ABB RobotStudio station: IRB1600_20220617-165440.rsstn

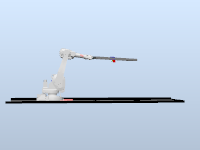
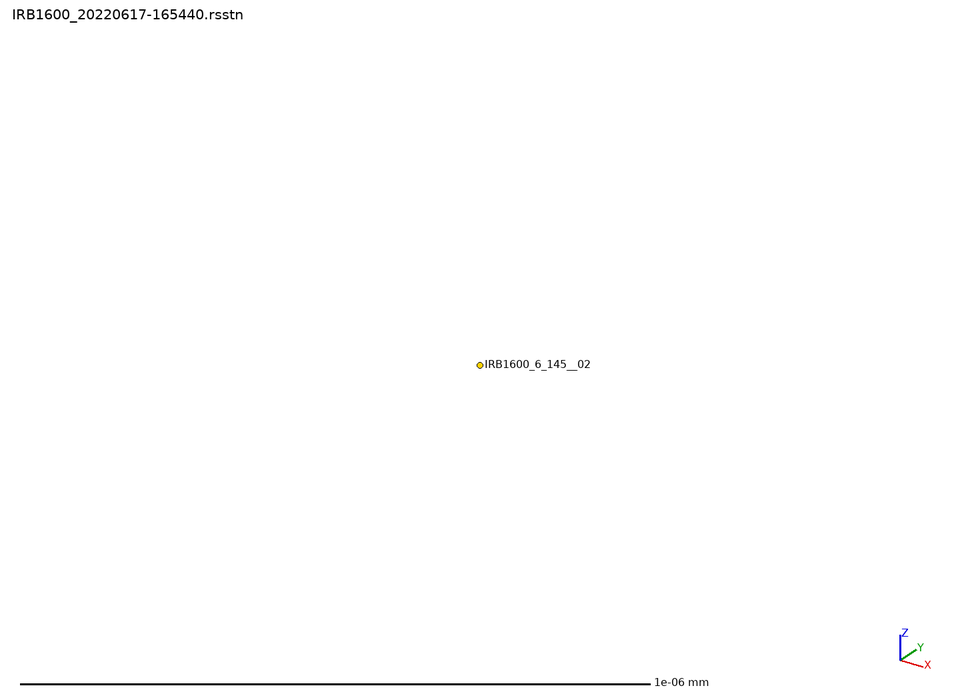
[picture v1: parts stored in the station drawn from their meshes, with robot base, taught points and paths (robot models come from the ABB library and are not in the file)]
Station Solution1 (saved by RobotStudio 22.1.9826.0)
Controller IRB1600_6_145
  mechanical unit ROB_1: IRB1600_6_145__02, 6 joints, base frame (0, 0, 0) mm
Layout (positions relative to the parent item):
  - IRB1600_6_145__02 [mechanism, from Robots\IRB1600_6_145_G_02.rslib] at (0, 0, 0) mm; joint values [0.0015, 0.282, -0.1091, -0.1819, -0.1284, 0.242] (rad or m)
  - flange_connector [part, from Tools\IsoPlate_small_Binzel.rslib] at (1000.78, 2.96, 1052.55) mm, rotated rx 126.74 ry 85.53 rz 128.07 deg
  - plane [part] at (1509.57, 17.68, 1033.56) mm, rotated rx 176.41 ry -2.67 rz -178.59 deg, size 1000 x 1000 x 50 mm
  - Frame_1 [frame]
  - Frame_2 [frame] at (-23.65, -1.83, 250.36) mm
Attachment: flange_connector is attached to IRB1600_6_145__02 / Link6
Attachment: plane is attached to flange_connector
Targets, tools, work objects and paths stored in the station, written as RAPID:
! task T_ROB1
MODULE Module1
  LOCAL PERS wobjdata egm_wobj:=[FALSE,TRUE,"",[[0,0,0],[1,0,0,0]],[[0,0,0],[1,0,0,0]]];
  PROC main()
    ConfJ \On;
  ENDPROC
  PROC EGM_CARTESIAN_MOVE()
    WaitTime 2;
  ENDPROC
  PROC RAPID_MOVE()
  ENDPROC
ENDMODULE

! task T_ROB1
MODULE CalibData
  TASK PERS tooldata Tooldata_4:=[TRUE,[[0,0,0],[1,0,0,0]],[1,[0,0,1],[1,0,0,0],0,0,0]];
  TASK PERS tooldata Tooldata_5:=[TRUE,[[0,0,0],[1,0,0,0]],[1,[0,0,1],[1,0,0,0],0,0,0]];
  TASK PERS tooldata Tooldata_6:=[TRUE,[[0,0,0],[1,0,0,0]],[1,[0,0,1],[1,0,0,0],0,0,0]];
  TASK PERS tooldata Tooldata_7:=[TRUE,[[-23.772999698,2.161000196,740.120999999],[0.707106781,0,-0.707106781,0]],[1,[0,0,1],[1,0,0,0],0,0,0]];
  TASK PERS wobjdata Workobject_2:=[FALSE,TRUE,"ROB_1",[[-55.133477186,-6.202200727,258.13059393],[1,0,0,0]],[[0,0,0],[1,0,0,0]]];
  TASK PERS tooldata Tooldata_9:=[TRUE,[[20.616002648,0.899999913,497.265999882],[0.707106781,-0.000000002,-0.707106781,0]],[1,[0,0,1],[1,0,0,0],0,0,0]];
ENDMODULE

